PROGRAM P0_01_Mapping
VAR
	
	AI_SPARE								:INT;
	DI_SPARE								:BOOL;
	AO_SPARE								:INT:=0;
	DO_SPARE								:BOOL:=FALSE;

	AI1										:ST_EL3174;
	AI2										:ST_EL3174;
	DI1										:ST_EL1819;
	DI2										:ST_EL1819;
	DI3										:ST_EL1819;
	DI4										:ST_EL1819;
	PS										:ST_EL9110;
	AO1										:ST_EL4124;
	AO2										:ST_EL4124;
	DO1										:ST_EL2809;
	DO2										:ST_EL2809;
	DO3										:ST_EL2809;
	DO4										:ST_EL2809;
	
	bIO_Card_Failure						:BOOL;

END_VAR

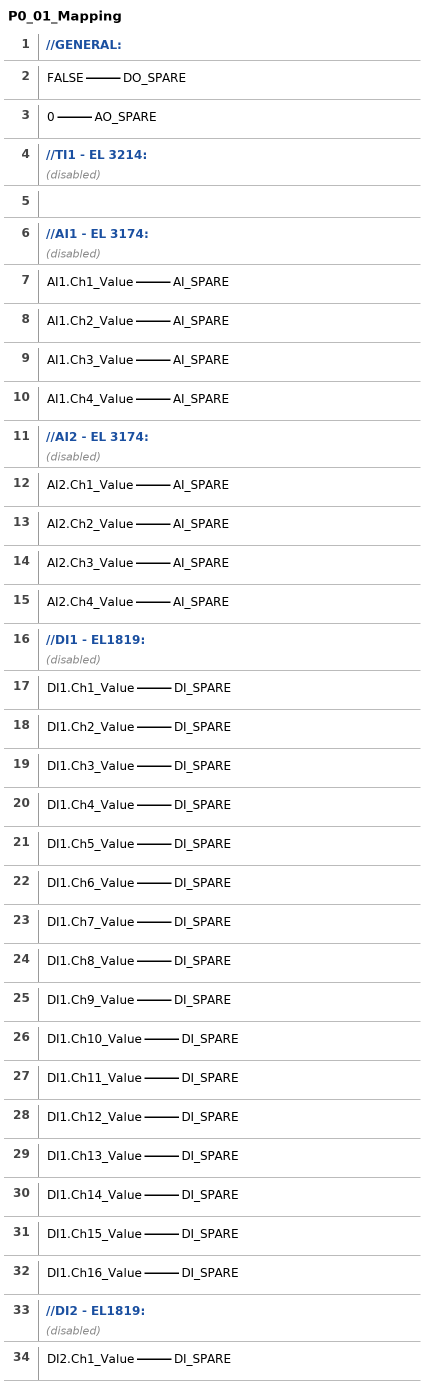
// NETWORK 1
// label: //GENERAL

// NETWORK 2
DO_SPARE := FALSE;

// NETWORK 3
AO_SPARE := 0;

// NETWORK 4 (disabled)
// label: //TI1 - EL 3214

// NETWORK 5

// NETWORK 6 (disabled)
// label: //AI1 - EL 3174

// NETWORK 7
AI_SPARE := AI1.Ch1_Value;

// NETWORK 8
AI_SPARE := AI1.Ch2_Value;

// NETWORK 9
AI_SPARE := AI1.Ch3_Value;

// NETWORK 10
AI_SPARE := AI1.Ch4_Value;

// NETWORK 11 (disabled)
// label: //AI2 - EL 3174

// NETWORK 12
AI_SPARE := AI2.Ch1_Value;

// NETWORK 13
AI_SPARE := AI2.Ch2_Value;

// NETWORK 14
AI_SPARE := AI2.Ch3_Value;

// NETWORK 15
AI_SPARE := AI2.Ch4_Value;

// NETWORK 16 (disabled)
// label: //DI1 - EL1819

// NETWORK 17
DI_SPARE := DI1.Ch1_Value;

// NETWORK 18
DI_SPARE := DI1.Ch2_Value;

// NETWORK 19
DI_SPARE := DI1.Ch3_Value;

// NETWORK 20
DI_SPARE := DI1.Ch4_Value;

// NETWORK 21
DI_SPARE := DI1.Ch5_Value;

// NETWORK 22
DI_SPARE := DI1.Ch6_Value;

// NETWORK 23
DI_SPARE := DI1.Ch7_Value;

// NETWORK 24
DI_SPARE := DI1.Ch8_Value;

// NETWORK 25
DI_SPARE := DI1.Ch9_Value;

// NETWORK 26
DI_SPARE := DI1.Ch10_Value;

// NETWORK 27
DI_SPARE := DI1.Ch11_Value;

// NETWORK 28
DI_SPARE := DI1.Ch12_Value;

// NETWORK 29
DI_SPARE := DI1.Ch13_Value;

// NETWORK 30
DI_SPARE := DI1.Ch14_Value;

// NETWORK 31
DI_SPARE := DI1.Ch15_Value;

// NETWORK 32
DI_SPARE := DI1.Ch16_Value;

// NETWORK 33 (disabled)
// label: //DI2 - EL1819

// NETWORK 34
DI_SPARE := DI2.Ch1_Value;

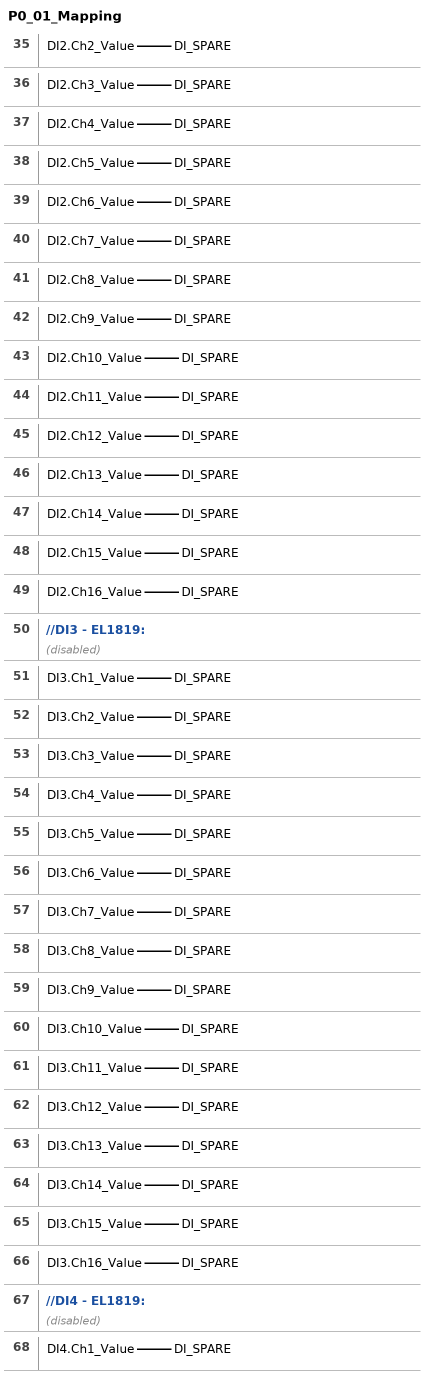
// NETWORK 35
DI_SPARE := DI2.Ch2_Value;

// NETWORK 36
DI_SPARE := DI2.Ch3_Value;

// NETWORK 37
DI_SPARE := DI2.Ch4_Value;

// NETWORK 38
DI_SPARE := DI2.Ch5_Value;

// NETWORK 39
DI_SPARE := DI2.Ch6_Value;

// NETWORK 40
DI_SPARE := DI2.Ch7_Value;

// NETWORK 41
DI_SPARE := DI2.Ch8_Value;

// NETWORK 42
DI_SPARE := DI2.Ch9_Value;

// NETWORK 43
DI_SPARE := DI2.Ch10_Value;

// NETWORK 44
DI_SPARE := DI2.Ch11_Value;

// NETWORK 45
DI_SPARE := DI2.Ch12_Value;

// NETWORK 46
DI_SPARE := DI2.Ch13_Value;

// NETWORK 47
DI_SPARE := DI2.Ch14_Value;

// NETWORK 48
DI_SPARE := DI2.Ch15_Value;

// NETWORK 49
DI_SPARE := DI2.Ch16_Value;

// NETWORK 50 (disabled)
// label: //DI3 - EL1819

// NETWORK 51
DI_SPARE := DI3.Ch1_Value;

// NETWORK 52
DI_SPARE := DI3.Ch2_Value;

// NETWORK 53
DI_SPARE := DI3.Ch3_Value;

// NETWORK 54
DI_SPARE := DI3.Ch4_Value;

// NETWORK 55
DI_SPARE := DI3.Ch5_Value;

// NETWORK 56
DI_SPARE := DI3.Ch6_Value;

// NETWORK 57
DI_SPARE := DI3.Ch7_Value;

// NETWORK 58
DI_SPARE := DI3.Ch8_Value;

// NETWORK 59
DI_SPARE := DI3.Ch9_Value;

// NETWORK 60
DI_SPARE := DI3.Ch10_Value;

// NETWORK 61
DI_SPARE := DI3.Ch11_Value;

// NETWORK 62
DI_SPARE := DI3.Ch12_Value;

// NETWORK 63
DI_SPARE := DI3.Ch13_Value;

// NETWORK 64
DI_SPARE := DI3.Ch14_Value;

// NETWORK 65
DI_SPARE := DI3.Ch15_Value;

// NETWORK 66
DI_SPARE := DI3.Ch16_Value;

// NETWORK 67 (disabled)
// label: //DI4 - EL1819

// NETWORK 68
DI_SPARE := DI4.Ch1_Value;

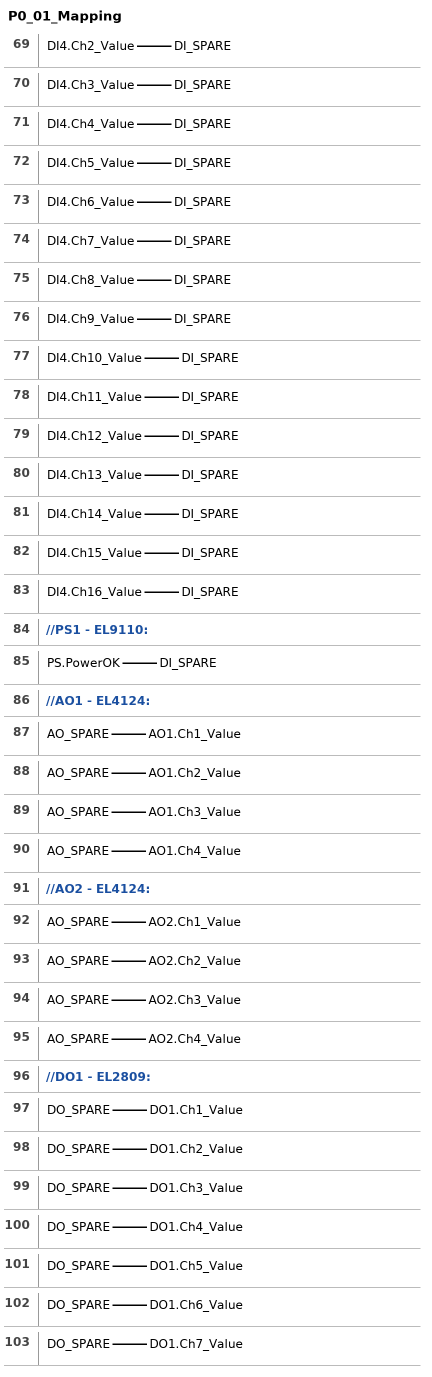
// NETWORK 69
DI_SPARE := DI4.Ch2_Value;

// NETWORK 70
DI_SPARE := DI4.Ch3_Value;

// NETWORK 71
DI_SPARE := DI4.Ch4_Value;

// NETWORK 72
DI_SPARE := DI4.Ch5_Value;

// NETWORK 73
DI_SPARE := DI4.Ch6_Value;

// NETWORK 74
DI_SPARE := DI4.Ch7_Value;

// NETWORK 75
DI_SPARE := DI4.Ch8_Value;

// NETWORK 76
DI_SPARE := DI4.Ch9_Value;

// NETWORK 77
DI_SPARE := DI4.Ch10_Value;

// NETWORK 78
DI_SPARE := DI4.Ch11_Value;

// NETWORK 79
DI_SPARE := DI4.Ch12_Value;

// NETWORK 80
DI_SPARE := DI4.Ch13_Value;

// NETWORK 81
DI_SPARE := DI4.Ch14_Value;

// NETWORK 82
DI_SPARE := DI4.Ch15_Value;

// NETWORK 83
DI_SPARE := DI4.Ch16_Value;

// NETWORK 84
// label: //PS1 - EL9110

// NETWORK 85
DI_SPARE := PS.PowerOK;

// NETWORK 86
// label: //AO1 - EL4124

// NETWORK 87
AO1.Ch1_Value := AO_SPARE;

// NETWORK 88
AO1.Ch2_Value := AO_SPARE;

// NETWORK 89
AO1.Ch3_Value := AO_SPARE;

// NETWORK 90
AO1.Ch4_Value := AO_SPARE;

// NETWORK 91
// label: //AO2 - EL4124

// NETWORK 92
AO2.Ch1_Value := AO_SPARE;

// NETWORK 93
AO2.Ch2_Value := AO_SPARE;

// NETWORK 94
AO2.Ch3_Value := AO_SPARE;

// NETWORK 95
AO2.Ch4_Value := AO_SPARE;

// NETWORK 96
// label: //DO1 - EL2809

// NETWORK 97
DO1.Ch1_Value := DO_SPARE;

// NETWORK 98
DO1.Ch2_Value := DO_SPARE;

// NETWORK 99
DO1.Ch3_Value := DO_SPARE;

// NETWORK 100
DO1.Ch4_Value := DO_SPARE;

// NETWORK 101
DO1.Ch5_Value := DO_SPARE;

// NETWORK 102
DO1.Ch6_Value := DO_SPARE;

// NETWORK 103
DO1.Ch7_Value := DO_SPARE;

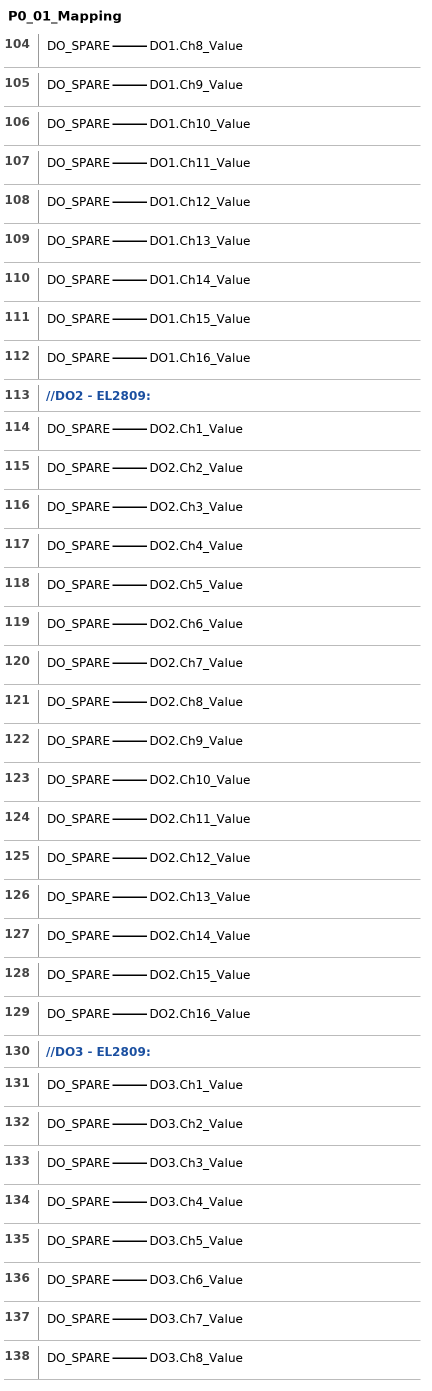
// NETWORK 104
DO1.Ch8_Value := DO_SPARE;

// NETWORK 105
DO1.Ch9_Value := DO_SPARE;

// NETWORK 106
DO1.Ch10_Value := DO_SPARE;

// NETWORK 107
DO1.Ch11_Value := DO_SPARE;

// NETWORK 108
DO1.Ch12_Value := DO_SPARE;

// NETWORK 109
DO1.Ch13_Value := DO_SPARE;

// NETWORK 110
DO1.Ch14_Value := DO_SPARE;

// NETWORK 111
DO1.Ch15_Value := DO_SPARE;

// NETWORK 112
DO1.Ch16_Value := DO_SPARE;

// NETWORK 113
// label: //DO2 - EL2809

// NETWORK 114
DO2.Ch1_Value := DO_SPARE;

// NETWORK 115
DO2.Ch2_Value := DO_SPARE;

// NETWORK 116
DO2.Ch3_Value := DO_SPARE;

// NETWORK 117
DO2.Ch4_Value := DO_SPARE;

// NETWORK 118
DO2.Ch5_Value := DO_SPARE;

// NETWORK 119
DO2.Ch6_Value := DO_SPARE;

// NETWORK 120
DO2.Ch7_Value := DO_SPARE;

// NETWORK 121
DO2.Ch8_Value := DO_SPARE;

// NETWORK 122
DO2.Ch9_Value := DO_SPARE;

// NETWORK 123
DO2.Ch10_Value := DO_SPARE;

// NETWORK 124
DO2.Ch11_Value := DO_SPARE;

// NETWORK 125
DO2.Ch12_Value := DO_SPARE;

// NETWORK 126
DO2.Ch13_Value := DO_SPARE;

// NETWORK 127
DO2.Ch14_Value := DO_SPARE;

// NETWORK 128
DO2.Ch15_Value := DO_SPARE;

// NETWORK 129
DO2.Ch16_Value := DO_SPARE;

// NETWORK 130
// label: //DO3 - EL2809

// NETWORK 131
DO3.Ch1_Value := DO_SPARE;

// NETWORK 132
DO3.Ch2_Value := DO_SPARE;

// NETWORK 133
DO3.Ch3_Value := DO_SPARE;

// NETWORK 134
DO3.Ch4_Value := DO_SPARE;

// NETWORK 135
DO3.Ch5_Value := DO_SPARE;

// NETWORK 136
DO3.Ch6_Value := DO_SPARE;

// NETWORK 137
DO3.Ch7_Value := DO_SPARE;

// NETWORK 138
DO3.Ch8_Value := DO_SPARE;

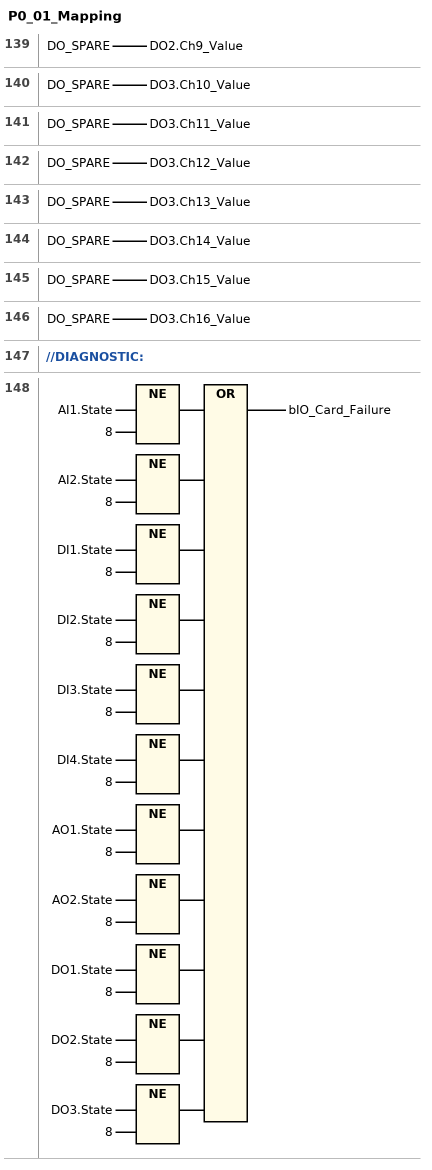
// NETWORK 139
DO2.Ch9_Value := DO_SPARE;

// NETWORK 140
DO3.Ch10_Value := DO_SPARE;

// NETWORK 141
DO3.Ch11_Value := DO_SPARE;

// NETWORK 142
DO3.Ch12_Value := DO_SPARE;

// NETWORK 143
DO3.Ch13_Value := DO_SPARE;

// NETWORK 144
DO3.Ch14_Value := DO_SPARE;

// NETWORK 145
DO3.Ch15_Value := DO_SPARE;

// NETWORK 146
DO3.Ch16_Value := DO_SPARE;

// NETWORK 147
// label: //DIAGNOSTIC

// NETWORK 148
bIO_Card_Failure := AI1.State <> 8 OR AI2.State <> 8 OR DI1.State <> 8 OR DI2.State <> 8 OR DI3.State <> 8 OR DI4.State <> 8 OR AO1.State <> 8 OR AO2.State <> 8 OR DO1.State <> 8 OR DO2.State <> 8 OR DO3.State <> 8;

END_PROGRAM

(* stored: Version 1.1.0.1, ProductVersion 3.1.4024.12
   POU P0_01_Mapping: Id {441d9743-fc60-4170-9c6f-0fd7cfda520a}, SpecialFunc None *)
